FUNCTION_BLOCK Grade_Mecanizada_Inovaisa (* Composite Function Block Type *)
  (* Standard: 61499-2 *)
  (* Version 0.0, 2/5/2026, Schneider Electric, template *)
  PACKAGE Hidryco.HidrycoLib;
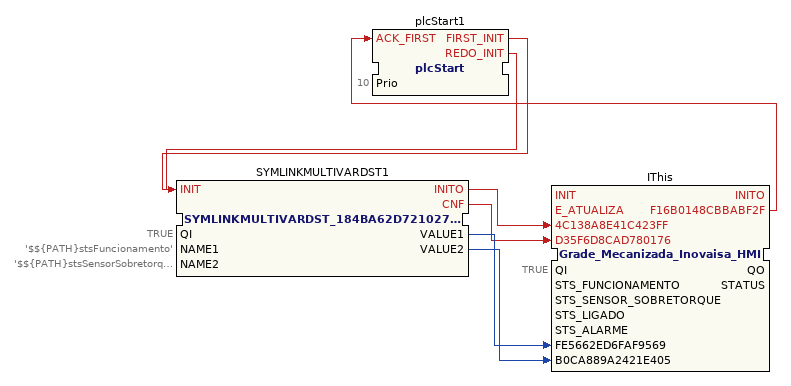
  FBS
    IThis : Grade_Mecanizada_Inovaisa_HMI(QI := TRUE);
    SYMLINKMULTIVARDST1 : SYMLINKMULTIVARDST_184BA62D721027C6E(QI := TRUE, NAME1 := '$${PATH}stsFuncionamento', NAME2 := '$${PATH}stsSensorSobretorque'); {SET_ATTRIBUTE(Configuration.GenericFBType.InterfaceParams, Runtime.System#I:=2;VALUE${I$}:INT,INT)}
    plcStart1 : plcStart(Prio := 10);
  END_FBS
  EVENT_CONNECTIONS
    plcStart1.FIRST_INIT TO SYMLINKMULTIVARDST1.INIT;
    plcStart1.REDO_INIT TO SYMLINKMULTIVARDST1.INIT;
    SYMLINKMULTIVARDST1.INITO TO IThis.4C138A8E41C423FF;
    SYMLINKMULTIVARDST1.CNF TO IThis.D35F6D8CAD780176;
    IThis.F16B0148CBBABF2F TO plcStart1.ACK_FIRST;
  END_CONNECTIONS
  DATA_CONNECTIONS
    SYMLINKMULTIVARDST1.VALUE1 TO IThis.FE5662ED6FAF9569;
    SYMLINKMULTIVARDST1.VALUE2 TO IThis.B0CA889A2421E405;
  END_CONNECTIONS
END_FUNCTION_BLOCK
